TYPE ST_LeakTester_CycleData :
STRUCT
	
	bPass							: BOOL;
	bFail							: BOOL;	

END_STRUCT
END_TYPE

(* stored: Version 1.1.0.1, ProductVersion 3.1.4026.17
   DUT ST_LeakTester_CycleData: Id {a87f5642-6635-4d10-aef6-f9a75b94d380} *)
